FUNCTION_BLOCK PUBLIC PAEEMotorFreqCtrl EXTENDS PAEEMotorBase
VAR_INPUT
END_VAR
VAR_OUTPUT
END_VAR
VAR
	_DesiredSpeed : LREAL;
	_ReqSpeed : LREAL;
	_Speed : LREAL;
	_VFDState : PANotifyState;
	_VFDStateACK : BOOL;
END_VAR

{attribute 'monitoring' := 'call'}
//{attribute 'TcRpcEnable'}
PROPERTY PUBLIC DesiredSpeed : LREAL
GET // PUBLIC
DesiredSpeed := _DesiredSpeed;
END_GET
SET // PUBLIC
_DesiredSpeed := DesiredSpeed;
Root.OnPropertyChangedLReal(THIS^, 43, _DesiredSpeed);
END_SET
END_PROPERTY

METHOD PUBLIC FB_postinit
VAR_INPUT
		root : IACVariobatch;
END_VAR
SUPER^.FB_postinit(root);  
root.OnPropertyChangedLReal(THIS^, 42, _Speed);
root.OnPropertyChangedLReal(THIS^, 43, _DesiredSpeed);
root.OnPropertyChangedInt(THIS^, 44, _VFDState);
root.OnPropertyChangedLReal(THIS^, 45, _ReqSpeed);
root.OnPropertyChangedBool(THIS^, 46, _VFDStateACK);
END_METHOD

METHOD PUBLIC InvokeSetterBool
VAR_INPUT
	PropertyID : INT;
	PropertyValue : BOOL;
END_VAR
SUPER^.InvokeSetterBool(PropertyID, PropertyValue);
CASE PropertyID OF
	46:
		VFDStateACK := PropertyValue;
END_CASE
END_METHOD

METHOD PUBLIC InvokeSetterEnum
VAR_INPUT
	PropertyID : INT;
	PropertyValue : INT;
END_VAR
SUPER^.InvokeSetterEnum(PropertyID, PropertyValue);
IF PropertyID = 44 THEN
	THIS^.VFDState := PropertyValue;
END_IF
END_METHOD

METHOD PUBLIC InvokeSetterLReal
VAR_INPUT
	PropertyID : INT;
	PropertyValue : LREAL;
END_VAR
SUPER^.InvokeSetterLReal(PropertyID, PropertyValue);
CASE PropertyID OF
	42:
		Speed := PropertyValue;
	43:
		DesiredSpeed := PropertyValue;
	45:
		ReqSpeed := PropertyValue;
END_CASE
END_METHOD

METHOD PUBLIC IsEnabledAcknowledgeAlarms : BOOL
VAR_INPUT
END_VAR
END_METHOD

METHOD OnInitMemory
VAR_INPUT
		root : IACVariobatch;
END_VAR
RegisterProperty(root, 42, GCL.cSizeLREAL); //Speed
RegisterProperty(root, 43, GCL.cSizeLREAL); //DesiredSpeed
RegisterProperty(root, 44, GCL.cSizeINT); //VFDState
RegisterProperty(root, 45, GCL.cSizeLREAL); //ReqSpeed
RegisterProperty(root, 46, GCL.cSizeBYTE); //VFDStateACK
SUPER^.OnInitMemory(root);
END_METHOD

METHOD PUBLIC OnSetVFDState
VAR_INPUT
END_VAR
END_METHOD

{attribute 'monitoring' := 'call'}
//{attribute 'TcRpcEnable'}
PROPERTY PUBLIC ReqSpeed : LREAL
GET // PUBLIC
ReqSpeed := _ReqSpeed;
END_GET
SET // PUBLIC
VAR
	_ReqPosition: LREAL;
END_VAR
_ReqSpeed := ReqSpeed;
Root.OnPropertyChangedLReal(THIS^, 45, _ReqSpeed);
IF Root.InSimulation THEN
	Speed := _ReqSpeed;
END_IF
END_SET
END_PROPERTY

{attribute 'monitoring' := 'call'}
//{attribute 'TcRpcEnable'}
PROPERTY PUBLIC Speed : LREAL
GET // PUBLIC
Speed := _Speed;
END_GET
SET // PUBLIC
_Speed := Speed;
Root.OnPropertyChangedLReal(THIS^, 42, _Speed);
END_SET
END_PROPERTY

{attribute 'monitoring' := 'call'}
//{attribute 'TcRpcEnable'}
PROPERTY PUBLIC VFDState : PANotifyState
GET // PUBLIC
VFDState := _VFDState;
END_GET
SET // PUBLIC
_VFDState := VFDState;
Root.OnPropertyChangedInt(THIS^, 44, _VFDState);
END_SET
END_PROPERTY

{attribute 'monitoring' := 'call'}
//{attribute 'TcRpcEnable'}
PROPERTY PUBLIC VFDStateACK : BOOL
GET // PUBLIC
VFDStateACK := _VFDStateACK;
END_GET
SET // PUBLIC
_VFDStateACK := VFDStateACK;
Root.OnPropertyChangedBool(THIS^, 46, _VFDStateACK);
END_SET
END_PROPERTY

END_FUNCTION_BLOCK

(* stored: Version 1.1.0.1, ProductVersion 3.1.4024.6
   POU PAEEMotorFreqCtrl: Id {c342ae5a-5ba3-49e2-9272-90e4166617b1}, SpecialFunc None
   Property DesiredSpeed: Id {ab266219-1df8-449c-9d3d-874ccb915e38}
   Get Get: Id {c105c40a-cde8-46a9-97e1-2c8db9468512}
   Set Set: Id {817509e2-67db-4555-82d9-db5b9e7bf58c}
   Method FB_postinit: Id {af7cc024-fb07-4644-b43a-52585d101b9b}
   Method InvokeSetterBool: Id {18667681-41ef-4d5c-bd2d-ecc9f0ed9eac}
   Method InvokeSetterEnum: Id {0dfd4823-267b-4d23-a9c8-28f19ebf302b}
   Method InvokeSetterLReal: Id {89ab80f7-996d-4e37-9f96-1a691c4abba8}
   Method IsEnabledAcknowledgeAlarms: Id {e4c41664-360a-4cdc-81c4-037be6f90cd6}
   Method OnInitMemory: Id {c706f7bf-e796-4956-9233-2ca06ca2970b}
   Method OnSetVFDState: Id {b996de8f-33d7-4d18-97b7-527ace2871fe}
   Property ReqSpeed: Id {3c801cdd-a6ce-4d7a-84ee-ff18852be388}
   Get Get: Id {58bdcbaa-2cbd-4e3f-bbe8-5101baf5dcf6}
   Set Set: Id {070b4b93-935c-46e8-9ad8-89c775c59ce9}
   Property Speed: Id {a15ae79a-83ba-455e-ba16-20a1af495cfe}
   Get Get: Id {b86f61b0-8153-4b28-9866-89bb3381b96e}
   Set Set: Id {f1c6e1bb-0737-4442-9a74-18cdad3ab454}
   Property VFDState: Id {8a91674c-e034-4200-8217-3a25e7a08444}
   Get Get: Id {bb1ab23d-30d3-4d25-a6a1-205fc358dfed}
   Set Set: Id {1a73b3c2-1649-4b3a-83f9-867b9fbb17e9}
   Property VFDStateACK: Id {8973d916-6413-4ede-b69c-e3587de65687}
   Get Get: Id {58e48fa3-d05c-4a39-91c9-899eea8e6464}
   Set Set: Id {be10bc28-ff5a-4d11-8c3e-6b5b26a0314b} *)
